# B&R Automation Studio project macie
Automation Studio 4.9

## Configuration Config1

### Hardware
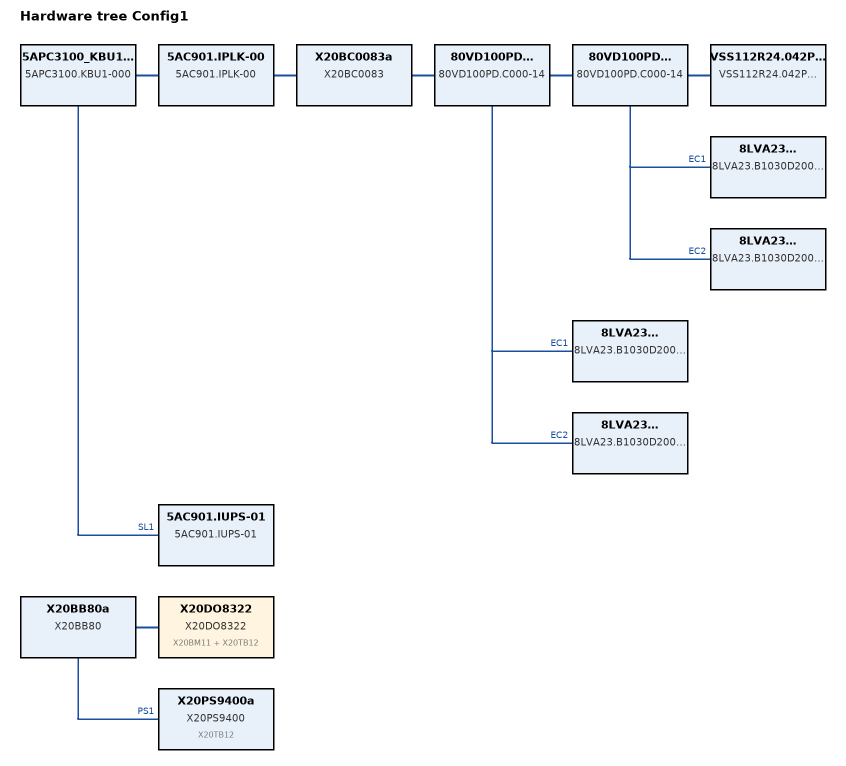
```
5AC901.IPLK-00 : 5AC901.IPLK-00 v1.8.0.1  [SL -> 5APC3100_KBU1_000.SL2]
  Connector IF1:
    MtuSize = 1500
    Channel1
    ChannelID1 = McAcpBroadcast
    ChannelType1 = OCTET[96]
    InternetAddress = 12.10.10.240
    SubnetMask = 255.255.255.0
5AC901.IUPS-01 : 5AC901.IUPS-01 v1.3.1.0  [SL -> 5APC3100_KBU1_000.SL1]
5APC3100_KBU1_000 : 5APC3100.KBU1-000 v2.2.1.0
  Connector IF3:
    AssignedOperatingSystem = ARemb
    ActivateDevice = 1
    Mode = Manual
    InternetAddress = 10.0.0.150
    SubnetMask = 255.255.255.0
    ActivateSnmp = 2
  Connector IF4:
    AssignedOperatingSystem = ARemb
    ActivateDevice = 1
    Mode = Manual
    InternetAddress = 192.168.0.20
    SubnetMask = 255.255.255.0
    ActivateSnmp = 2
  Connector IF5:
    AssignedOperatingSystem = ARemb
  Connector IF6:
    AssignedOperatingSystem = ARemb
  Connector IF7:
    AssignedOperatingSystem = ARemb
  Connector IF8:
    AssignedOperatingSystem = ARemb
  ConfigurationID = prawdziwaDelta_Config1
  Simulation = 1
  TimerDeviceType = EPLX2X
  TimerDevice = 5AC901.IPLK-00.IF1
  TaskClassIdleTime = 2000
  Cyclic1Tolerance = 0
  FileDevice1
  FileDeviceName1 = CNC_PrgDir
  FileDevicePath1 = C:\projects\CNC_PrgDir
  ActivateOpcUa = 1
  OpcUaInformationModels_PV_Version = 1
80VD100PD.C000-14 : 80VD100PD.C000-14 v2.5.0.0  [PLK1 -> X20BC0083a.PLK2 (NodeNumber=1) [Cable Type=PowerlinkCable, Length=10, Version=1.0.0.3]; PLK2 -> 80VD100PD.C000-14a.PLK1 (NodeNumber=1) [Cable Type=PowerlinkCable, Length=10, Version=1.0.0.3]; EC1 -> 8LVA23.B1030D200-0.EC; EC2 -> 8LVA23.B1030D200-0a.EC; MT2 -> 8LVA23.B1030D200-0a.MT]
  DriveConfiguration/Module:
    McAcoposTypeID = AcoposMicroDConfig
    ActivateACOPOSSimulationOnPLC = 0
  DriveConfiguration/Channel[1]/RealAxis:
    AxisReference = gAxisQ1
    MechanicalElementsIsInvisible = 0
  DriveConfiguration/Channel[1]/RealAxis/MechanicalElements/Gearbox:
    InputIsReadOnly = 0
    Input = 25
    OutputIsReadOnly = 0
    Output = 1
  DriveConfiguration/Channel[1]/RealAxis/MechanicalElements/RotaryToLinearTransformation:
    ReferenceDistanceIsReadOnly = 0
    ReferenceDistance = 1
  DriveConfiguration/Channel[1]/RealAxis/Controller:
    ModeIsReadOnly = 0
    Mode = PositionController
  DriveConfiguration/Channel[1]/RealAxis/Controller/Mode/Position:
    ProportionalGain = 402
    IntegrationTime = 0.0
    PredictionTime = 0.0004
    TotalDelayTime = 0.0004
  DriveConfiguration/Channel[1]/RealAxis/Controller/Mode/Speed:
    ProportionalGainIsReadOnly = 0
    ProportionalGain = 1.7
    IntegrationTimeIsReadOnly = 0
    IntegrationTime = 0.0
    FilterTimeIsReadOnly = 0
    FilterTime = 0.0
  DriveConfiguration/Channel[1]/RealAxis/Controller/Mode/LoopFilters:
    LoopFilterXIsReadOnly = 0
    LoopFilter1 = NotUsed
    LoopFilter2 = NotUsed
    LoopFilter3 = NotUsed
  DriveConfiguration/Channel[1]/RealAxis/Homing:
    ModeIsReadOnly = 0
    Mode = Absolute
  DriveConfiguration/Channel[1]/RealAxis/Homing/Mode:
    Position = 0
  DriveConfiguration/Channel[1]/RealAxis/Homing:
    RestorePositionVariable = 
  DriveConfiguration/Channel[1]/RealAxis/StopReaction:
    QuickstopIsReadOnly = 0
    Quickstop = DecelerationLimit
    DriveErrorIsReadOnly = 0
    DriveError = DecelerationLimit
  DriveConfiguration/Channel[1]/RealAxis/MovementErrorLimits:
    PositionError = 1.0
    VelocityErrorMonitoring = Automatic1
  DriveConfiguration/Channel[1]/RealAxis:
    JerkFilterIsReadOnly = 0
    JerkFilter = NotUsed
    ZeroVibrationFilter = NotUsed
  DriveConfiguration/Channel[1]/RealAxis/DigitalInputs/HomingSwitch:
    SourceIsReadOnly = 0
    Source = NotUsed
    Level = High
  DriveConfiguration/Channel[1]/RealAxis/DigitalInputs/PositiveLimitSwitch:
    SourceIsReadOnly = 0
    Source = NotUsed
    Level = High
  DriveConfiguration/Channel[1]/RealAxis/DigitalInputs/NegativeLimitSwitch:
    SourceIsReadOnly = 0
    Source = NotUsed
    Level = High
  DriveConfiguration/Channel[1]/RealAxis/DigitalInputs/Trigger1:
    Source = X2Trigger1
    Level = High
  DriveConfiguration/Channel[1]/RealAxis/DigitalInputs/Trigger2:
    Source = X2Trigger2
    Level = High
  DriveConfiguration/Channel[1]/RealAxis/DigitalInputs/Quickstop:
    Input = Trigger2
  DriveConfiguration/Channel[1]/RealAxis/Simulation:
    SimulationModeOnPLC = SetValueGeneration
    SimulationModeOnACOPOS = NotUsed
  DriveConfiguration/Channel[1]:
    ExternalEncoderAxis = NotUsed
  DriveConfiguration/Channel[2]/RealAxis:
    AxisReference = gAxisQ2
    MechanicalElementsIsInvisible = 0
  DriveConfiguration/Channel[2]/RealAxis/MechanicalElements/Gearbox:
    InputIsReadOnly = 0
    Input = 25
    OutputIsReadOnly = 0
    Output = 1
  DriveConfiguration/Channel[2]/RealAxis/MechanicalElements/RotaryToLinearTransformation:
    ReferenceDistanceIsReadOnly = 0
    ReferenceDistance = 1
  DriveConfiguration/Channel[2]/RealAxis/Controller:
    ModeIsReadOnly = 0
    Mode = PositionController
  DriveConfiguration/Channel[2]/RealAxis/Controller/Mode/Position:
    ProportionalGain = 393
    IntegrationTime = 0.0
    PredictionTime = 0.0004
    TotalDelayTime = 0.0004
  DriveConfiguration/Channel[2]/RealAxis/Controller/Mode/Speed:
    ProportionalGainIsReadOnly = 0
    ProportionalGain = 1.65
    IntegrationTimeIsReadOnly = 0
    IntegrationTime = 0.0
    FilterTimeIsReadOnly = 0
    FilterTime = 0.0
  DriveConfiguration/Channel[2]/RealAxis/Controller/Mode/LoopFilters:
    LoopFilterXIsReadOnly = 0
    LoopFilter1 = NotUsed
    LoopFilter2 = NotUsed
    LoopFilter3 = NotUsed
  DriveConfiguration/Channel[2]/RealAxis/Homing:
    ModeIsReadOnly = 0
    Mode = Absolute
  DriveConfiguration/Channel[2]/RealAxis/Homing/Mode:
    Position = 0
  DriveConfiguration/Channel[2]/RealAxis/Homing:
    RestorePositionVariable = 
  DriveConfiguration/Channel[2]/RealAxis/StopReaction:
    QuickstopIsReadOnly = 0
    Quickstop = DecelerationLimit
    DriveErrorIsReadOnly = 0
    DriveError = DecelerationLimit
  DriveConfiguration/Channel[2]/RealAxis/MovementErrorLimits:
    PositionError = 1.0
    VelocityErrorMonitoring = Automatic1
  DriveConfiguration/Channel[2]/RealAxis:
    JerkFilterIsReadOnly = 0
    JerkFilter = NotUsed
    ZeroVibrationFilter = NotUsed
  DriveConfiguration/Channel[2]/RealAxis/DigitalInputs/HomingSwitch:
    SourceIsReadOnly = 0
    Source = NotUsed
    Level = High
  DriveConfiguration/Channel[2]/RealAxis/DigitalInputs/PositiveLimitSwitch:
    SourceIsReadOnly = 0
    Source = NotUsed
    Level = High
  DriveConfiguration/Channel[2]/RealAxis/DigitalInputs/NegativeLimitSwitch:
    SourceIsReadOnly = 0
    Source = NotUsed
    Level = High
  DriveConfiguration/Channel[2]/RealAxis/DigitalInputs/Trigger1:
    Source = X2Trigger1
    Level = High
  DriveConfiguration/Channel[2]/RealAxis/DigitalInputs/Trigger2:
    Source = X2Trigger2
    Level = High
  DriveConfiguration/Channel[2]/RealAxis/DigitalInputs/Quickstop:
    Input = Trigger2
  DriveConfiguration/Channel[2]/RealAxis/Simulation:
    SimulationModeOnPLC = SetValueGeneration
    SimulationModeOnACOPOS = NotUsed
  DriveConfiguration/Channel[2]:
    ExternalEncoderAxis = NotUsed
80VD100PD.C000-14a : 80VD100PD.C000-14 v2.5.0.0  [PLK1 -> 80VD100PD.C000-14.PLK2 (NodeNumber=2) [Cable Type=PowerlinkCable, Length=10, Version=1.0.0.3]; PLK2 -> VSS112R24.042P-000.PLK1 (NodeNumber=2) [Cable Type=PowerlinkCable, Length=10, Version=1.0.0.3]; EC1 -> 8LVA23.B1030D200-0b.EC; EC2 -> 8LVA23.B1030D200-0c.EC; MT2 -> 8LVA23.B1030D200-0c.MT]
  DriveConfiguration/Module:
    McAcoposTypeID = AcoposMicroDConfig
    ActivateACOPOSSimulationOnPLC = 0
  DriveConfiguration/Channel[1]/RealAxis:
    AxisReference = gAxisQ3
    MechanicalElementsIsInvisible = 0
  DriveConfiguration/Channel[1]/RealAxis/MechanicalElements/Gearbox:
    InputIsReadOnly = 0
    Input = 25
    OutputIsReadOnly = 0
    Output = 1
  DriveConfiguration/Channel[1]/RealAxis/MechanicalElements/RotaryToLinearTransformation:
    ReferenceDistanceIsReadOnly = 0
    ReferenceDistance = 1
  DriveConfiguration/Channel[1]/RealAxis/Controller:
    ModeIsReadOnly = 0
    Mode = PositionController
  DriveConfiguration/Channel[1]/RealAxis/Controller/Mode/Position:
    ProportionalGain = 400
    IntegrationTime = 0.0
    PredictionTime = 0.0004
    TotalDelayTime = 0.0004
  DriveConfiguration/Channel[1]/RealAxis/Controller/Mode/Speed:
    ProportionalGainIsReadOnly = 0
    ProportionalGain = 1.7
    IntegrationTimeIsReadOnly = 0
    IntegrationTime = 0.0
    FilterTimeIsReadOnly = 0
    FilterTime = 0.0
  DriveConfiguration/Channel[1]/RealAxis/Controller/Mode/LoopFilters:
    LoopFilterXIsReadOnly = 0
    LoopFilter1 = NotUsed
    LoopFilter2 = NotUsed
    LoopFilter3 = NotUsed
  DriveConfiguration/Channel[1]/RealAxis/Homing:
    ModeIsReadOnly = 0
    Mode = Absolute
  DriveConfiguration/Channel[1]/RealAxis/Homing/Mode:
    Position = 0
  DriveConfiguration/Channel[1]/RealAxis/Homing:
    RestorePositionVariable = 
  DriveConfiguration/Channel[1]/RealAxis/StopReaction:
    QuickstopIsReadOnly = 0
    Quickstop = DecelerationLimit
    DriveErrorIsReadOnly = 0
    DriveError = DecelerationLimit
  DriveConfiguration/Channel[1]/RealAxis/MovementErrorLimits:
    PositionError = 1.0
    VelocityErrorMonitoring = Automatic1
  DriveConfiguration/Channel[1]/RealAxis:
    JerkFilterIsReadOnly = 0
    JerkFilter = NotUsed
    ZeroVibrationFilter = NotUsed
  DriveConfiguration/Channel[1]/RealAxis/DigitalInputs/HomingSwitch:
    SourceIsReadOnly = 0
    Source = NotUsed
    Level = High
  DriveConfiguration/Channel[1]/RealAxis/DigitalInputs/PositiveLimitSwitch:
    SourceIsReadOnly = 0
    Source = NotUsed
    Level = High
  DriveConfiguration/Channel[1]/RealAxis/DigitalInputs/NegativeLimitSwitch:
    SourceIsReadOnly = 0
    Source = NotUsed
    Level = High
  DriveConfiguration/Channel[1]/RealAxis/DigitalInputs/Trigger1:
    Source = X2Trigger1
    Level = High
  DriveConfiguration/Channel[1]/RealAxis/DigitalInputs/Trigger2:
    Source = X2Trigger2
    Level = High
  DriveConfiguration/Channel[1]/RealAxis/DigitalInputs/Quickstop:
    Input = Trigger2
  DriveConfiguration/Channel[1]/RealAxis/Simulation:
    SimulationModeOnPLC = SetValueGeneration
    SimulationModeOnACOPOS = NotUsed
  DriveConfiguration/Channel[1]:
    ExternalEncoderAxis = NotUsed
  DriveConfiguration/Channel[2]/RealAxis:
    AxisReference = gAxis_1
    MechanicalElementsIsInvisible = 0
  DriveConfiguration/Channel[2]/RealAxis/MechanicalElements/Gearbox:
    InputIsReadOnly = 0
    Input = 1
    OutputIsReadOnly = 0
    Output = 1
  DriveConfiguration/Channel[2]/RealAxis/MechanicalElements/RotaryToLinearTransformation:
    ReferenceDistanceIsReadOnly = 0
    ReferenceDistance = 1
  DriveConfiguration/Channel[2]/RealAxis/Controller:
    ModeIsReadOnly = 0
    Mode = PositionController
  DriveConfiguration/Channel[2]/RealAxis/Controller/Mode/Position:
    ProportionalGain = 50.0
    IntegrationTime = 0.0
    PredictionTime = 0.0004
    TotalDelayTime = 0.0004
  DriveConfiguration/Channel[2]/RealAxis/Controller/Mode/Speed:
    ProportionalGainIsReadOnly = 0
    ProportionalGain = 2.0
    IntegrationTimeIsReadOnly = 0
    IntegrationTime = 0.0
    FilterTimeIsReadOnly = 0
    FilterTime = 0.0
  DriveConfiguration/Channel[2]/RealAxis/Controller/Mode/LoopFilters:
    LoopFilterXIsReadOnly = 0
    LoopFilter1 = NotUsed
    LoopFilter2 = NotUsed
    LoopFilter3 = NotUsed
  DriveConfiguration/Channel[2]/RealAxis/Homing:
    ModeIsReadOnly = 0
    Mode = Direct
  DriveConfiguration/Channel[2]/RealAxis/Homing/Mode:
    Position = 0.0
    ReferencePulse = NotUsed
  DriveConfiguration/Channel[2]/RealAxis/Homing:
    RestorePositionVariable = 
  DriveConfiguration/Channel[2]/RealAxis/StopReaction:
    QuickstopIsReadOnly = 0
    Quickstop = DecelerationLimit
    DriveErrorIsReadOnly = 0
    DriveError = DecelerationLimit
  DriveConfiguration/Channel[2]/RealAxis/MovementErrorLimits:
    PositionError = 1.0
    VelocityErrorMonitoring = Automatic1
  DriveConfiguration/Channel[2]/RealAxis:
    JerkFilterIsReadOnly = 0
    JerkFilter = NotUsed
    ZeroVibrationFilter = NotUsed
  DriveConfiguration/Channel[2]/RealAxis/DigitalInputs/HomingSwitch:
    SourceIsReadOnly = 0
    Source = NotUsed
    Level = High
  DriveConfiguration/Channel[2]/RealAxis/DigitalInputs/PositiveLimitSwitch:
    SourceIsReadOnly = 0
    Source = NotUsed
    Level = High
  DriveConfiguration/Channel[2]/RealAxis/DigitalInputs/NegativeLimitSwitch:
    SourceIsReadOnly = 0
    Source = NotUsed
    Level = High
  DriveConfiguration/Channel[2]/RealAxis/DigitalInputs/Trigger1:
    Source = X2Trigger1
    Level = High
  DriveConfiguration/Channel[2]/RealAxis/DigitalInputs/Trigger2:
    Source = X2Trigger2
    Level = High
  DriveConfiguration/Channel[2]/RealAxis/DigitalInputs/Quickstop:
    Input = Trigger2
  DriveConfiguration/Channel[2]/RealAxis/Simulation:
    SimulationModeOnPLC = SetValueGeneration
    SimulationModeOnACOPOS = NotUsed
  DriveConfiguration/Channel[2]:
    ExternalEncoderAxis = NotUsed
8LVA23.B1030D200-0 : 8LVA23.B1030D200-0 v2.2.0.3  [EC -> 80VD100PD.C000-14.EC1; MT -> 80VD100PD.C000-14.MT1]
  M1/MotorParameters:
    MOTOR_AMB_TEMP_RATED = 40
8LVA23.B1030D200-0a : 8LVA23.B1030D200-0 v2.2.0.3  [EC -> 80VD100PD.C000-14.EC2; MT -> 80VD100PD.C000-14.MT2]
  M1/MotorParameters:
    MOTOR_AMB_TEMP_RATED = 40
8LVA23.B1030D200-0b : 8LVA23.B1030D200-0 v2.2.0.3  [EC -> 80VD100PD.C000-14a.EC1; MT -> 80VD100PD.C000-14a.MT1]
  M1/MotorParameters:
    MOTOR_AMB_TEMP_RATED = 40
8LVA23.B1030D200-0c : 8LVA23.B1030D200-0 v2.2.0.3  [EC -> 80VD100PD.C000-14a.EC2; MT -> 80VD100PD.C000-14a.MT2]
  M1/MotorParameters:
    MOTOR_AMB_TEMP_RATED = 40
VSS112R24.042P-000 : VSS112R24.042P-000 v1.9.0.730  [PLK1 -> 80VD100PD.C000-14a.PLK2 (NodeNumber=4) [Cable Type=PowerlinkCable, Length=10, Version=1.0.0.3]]
  Supervision = off
  VisionConfig = gCamera
X20BB80a : X20BB80 v1.1.0.0
X20BC0083a : X20BC0083 v2.14.0.0  [PLK1 -> 5AC901.IPLK-00.IF1 (NodeNumber=3) [Cable Type=PowerlinkCable, Length=10, Version=1.0.0.3]; PLK2 -> 80VD100PD.C000-14.PLK1 (NodeNumber=3) [Cable Type=PowerlinkCable, Length=10, Version=1.0.0.3]; SL -> X20BB80a.SL1]
  Supervision = off
X20BM11a : X20BM11 v1.1.0.0  [X2X1 -> X20BB80a.IF1]
X20DO8322 : X20DO8322 v1.5.0.0  [SS1 -> X20TB12b.SS; SL -> X20BM11a.SL1]
X20PS9400a : X20PS9400 v1.8.0.0  [SS1 -> X20TB12a.SS; PS -> X20BB80a.PS1]
  Supervision = off
X20TB12a : X20TB12 v1.0.0.0
X20TB12b : X20TB12 v1.0.0.0
```

### Config_8.pickregister - 5APC3100_KBU1_000/mappMotion/Config_8.pickregister
```
Element gPickRegister (Type=pickregister)
  Type = LinearConveyor
    StandardFrameName = ConveyorPick
    Length = 600
    Width = 120
    Height = 6
    MaxPositionError = 10
    MotionSource = Axis
      AxisRef = gAxis_1
      MovementLimits = UseAxisLimits
        Direction = Bidirectional
  SceneViewerObject = Used
    VisualRepresentation = Conveyor belt
      Dimensions:
        Length = 0.0
        Width = 0.0
        Height = 0.0
      Translation:
        X = 0.0
        Y = 0.0
        Z = 0.0
      Orientation:
        Angle1 = 0.0
        Angle2 = 0.0
        Angle3 = 0.0
    Content:
      Template[1]:
        VisualRepresentation = 2DShape
          ShapeType:
            Dimensions:
              Radius = 25.0
            Translation:
              X = 0.0
              Y = 0.0
              Z = 0.0
            Orientation:
              Angle1 = 0.0
              Angle2 = 0.0
              Angle3 = 0.0
        Filter:
          ObjectState:
            State[1] = 1
      Template[2]:
        VisualRepresentation:
          Size = 50.0
        Filter:
          ObjectState:
            State[1] = 2
  Alarms = None
Element gPlaceRegister (Type=pickregister)
  Type = LinearConveyor
    StandardFrameName = ConveyorPlace
    Length = 215
    Width = 60
    Height = 10
    MaxItems = 5
    MaxPositionError = 10
    MotionSource = Axis
      AxisRef = gAxis_2
      MovementLimits = UseAxisLimits
        Direction = Bidirectional
  SceneViewerObject = Used
    VisualRepresentation = Cuboid
      Dimensions:
        Length = 215
        Width = 60
        Height = 50
      Translation:
        X = 0.0
        Y = 0.0
        Z = 0.0
      Orientation:
        Angle1 = 0.0
        Angle2 = 0.0
        Angle3 = 0.0
    Content:
      Template[1]:
        VisualRepresentation = 2DShape
          ShapeType:
            Dimensions:
              Radius = 25.0
            Translation:
              X = 0.0
              Y = 0.0
              Z = 0.0
            Orientation:
              Angle1 = 0.0
              Angle2 = 0.0
              Angle3 = 0.0
        Filter:
          ObjectState:
            State[1] = 1
      Template[2]:
        VisualRepresentation:
          Size = 50.0
        Filter:
          ObjectState:
            State[1] = 1
  Alarms = None
```

## Logical view

### Robotic.st
```iecst
VAR CONSTANT
P1 : McPointType := (Pos:=(X:=0, Y:=0, Z:=-650));
P2 : McPointType := (Pos:=(X:=-50, Y:=-20, Z:=-600));
P0 : McPointType := (Pos:=(X:=0, Y:=0, Z:=-560));
	END_VAR

	PROGRAM _MAIN
	Feedrate(5000);   //move with reduced speed
	MoveJ(P1);        //move system to point P1
	MoveJ(P2);        //move system to point P2

	WaitTime(3);        //wait for 3 seconds

	MoveJ(P0);        //move back to origin position
	END_PROGRAM
```

### Program Logical/PickAndPlace/PrgMechs (IEC) - Handle Delta & Conveyor Belts

#### Main.st
```iecst
PROGRAM _INIT

	MpDelta4Axis_0.Override := 100.0;
	MpDelta4Axis_0.Enable   := TRUE;

	AxisParameters_0.Velocity     := 50.0;
	AxisParameters_0.Acceleration := 50.0;
	AxisParameters_0.Deceleration := 50.0;

	AxisParameters_1.Velocity     := 130.0;
	AxisParameters_1.Acceleration := 50.0;
	AxisParameters_1.Deceleration := 50.0;

	MpAxisBasic_0.Enable := TRUE;
	MpAxisBasic_1.Enable := TRUE;

	// dummy call of axis PVs just to avoid warning -2141192189 "The PV 'gAxisQx' does not exists" in logger
	gAxisQ1;
	gAxisQ2;
	gAxisQ3;
	gAxisQ4;

END_PROGRAM

PROGRAM _CYCLIC

    (* Prepare mechanics: Robot & conveyors *)
	CASE RC_Step OF

		(* first preparing robot *)
		RC_WAIT_ENABLE:
			IF MpDelta4Axis_0.Active THEN
				RC_Step := RC_POWER_ROBOT;
			END_IF

		RC_POWER_ROBOT:
			MpDelta4Axis_0.Power := TRUE;
			IF MpDelta4Axis_0.PowerOn THEN
				RC_Step := RC_HOME_ROBOT;
			END_IF

		RC_HOME_ROBOT:
			MpDelta4Axis_0.Home := TRUE;
			IF MpDelta4Axis_0.IsHomed THEN
				MpDelta4Axis_0.Home := FALSE;
				RC_Step := RC_ROBOT_READY;
			END_IF

		RC_ROBOT_READY:
			RC_Step := RC_WAIT_ENABLE_AXIS_FB;

			(* preparing conveyors *)
		RC_WAIT_ENABLE_AXIS_FB:
			IF MpAxisBasic_0.Active THEN
				IF MpAxisBasic_1.Active THEN
					RC_Step := RC_POWER_AXIS;
				END_IF
			ELSIF MpAxisBasic_0.Error  THEN
				LastStep := RC_Step;
				RC_Step  := RC_ERROR;
			END_IF;

		RC_POWER_AXIS:
			MpAxisBasic_0.Power := TRUE;
			MpAxisBasic_1.Power := TRUE;
			RC_Step := RC_WAIT_POWER_AXIS;

		RC_WAIT_POWER_AXIS:
			IF MpAxisBasic_0.PowerOn THEN
				IF MpAxisBasic_1.PowerOn THEN
					RC_Step := RC_HOME_AXIS;
				END_IF
			ELSIF MpAxisBasic_0.Error  THEN
				LastStep := RC_Step;
				RC_Step  := RC_ERROR;
			END_IF;

		RC_HOME_AXIS:
			MpAxisBasic_0.Home := TRUE;
			MpAxisBasic_1.Home := TRUE;
			RC_Step := RC_WAIT_HOME_AXIS;

		RC_WAIT_HOME_AXIS:
			IF MpAxisBasic_0.IsHomed THEN
				IF MpAxisBasic_0.IsHomed THEN
					MpAxisBasic_0.Home := FALSE;
					MpAxisBasic_1.Home := FALSE;
					RC_Step := RC_READY;
				END_IF
			ELSIF MpAxisBasic_0.Error  THEN
				LastStep := RC_Step;
				RC_Step  := RC_ERROR;
			END_IF;

		RC_READY:
			ReadyMechanics := TRUE;
			IF CmdStart AND ReadyToStart THEN
				RC_Step := RC_START_PROCESS;
			END_IF;

			(* start conveyors to move *)
		RC_START_PROCESS:
			MpAxisBasic_0.MoveVelocity := TRUE;
			//  MpAxisBasic_1.MoveVelocity := TRUE;
			RC_Step := RC_WAIT_PROCESS_STARTED;

		RC_WAIT_PROCESS_STARTED:
			IF MpAxisBasic_0.Info.PLCopenState = mcAXIS_CONTINUOUS_MOTION THEN
				//   IF MpAxisBasic_1.Info.PLCopenState = mcAXIS_CONTINUOUS_MOTION THEN
				RC_Step := RC_PROCESSING;
				//  END_IF
			ELSIF MpAxisBasic_0.Error  THEN
				LastStep := RC_Step;
				RC_Step  := RC_ERROR;
			END_IF;

		RC_PROCESSING:
			IF MpAxisBasic_0.Error  THEN
				LastStep := RC_Step;
				RC_Step  := RC_ERROR;
			END_IF;

		RC_ERROR:
			ReadyMechanics := FALSE;

	END_CASE

	ReadyToStart := ReadyMechanics AND ReadyPickReg AND ReadyPlaceReg AND ReadyPickCore;

	(* Call FBs *)
	MpDelta4Axis_0.MpLink     := ADR(g4AxDeltaA);
	MpDelta4Axis_0.Parameters := ADR(DeltaParameters);
	MpDelta4Axis_0();

	MpAxisBasic_0.MpLink     := ADR(gAxis_1);
	MpAxisBasic_0.Parameters := ADR(AxisParameters_0);
	MpAxisBasic_0();

	MpAxisBasic_1.MpLink     := ADR(gAxis_2);
	MpAxisBasic_1.Parameters := ADR(AxisParameters_1);
	MpAxisBasic_1();

	PickConveyorPosition  := MpAxisBasic_0.Position;
	PlaceConveyorPosition := MpAxisBasic_1.Position;

END_PROGRAM
```

### Program Logical/PickAndPlace/PrgPlace (IEC) - Place the products

#### Types.typ
```iecst
TYPE
	PlaceStepEnum :
		(
		P_WAIT_ENABLE,
		P_ENABLE_REGISTER_FB,
		P_WAIT_ENABLE_REGISTER_FB,
		P_ENABLE_REGISTER_COMP,
		P_WAIT_ENABLE_REGISTER_COMP,
		P_ENABLE_ADD_REGISTER_FBS,
		P_WAIT_ENABLE_ADD_REGISTER_FBS,
		P_WAIT_START_PROCESS,
		P_CREATE_OBJECTS,
		P_WAIT_CREATE_OBJECTS,
		P_WAIT_REGISTER_FULL,
		P_DELAY_DELETE,
		P_DELETE_OBJECTS,
		P_WAIT_DELETE_OBJECTS,
		P_DELAY_CREATE,
		P_ERROR
	);
END_TYPE
```

#### Variables.var
```iecst
VAR
	P_Step : PlaceStepEnum;
	LastStep : PlaceStepEnum;
	Error : BOOL;
	PlaceHoldersSpacing : LREAL;
	LastPlaceHolderConveyorPosition : LREAL;
	ElapsedDistance : LREAL;
END_VAR
(*   *)
(*Functionblocks*)
VAR
	MpPickRegCreatePlaceholder1 : MpPickRegCreateObject;
	MpPickRegCreatePlaceholder2 : MpPickRegCreateObject;
	MpPickRegCreatePlaceholder3 : MpPickRegCreateObject;
	MpPickRegCreatePlaceholder : MpPickRegCreateObject;
	MpPickRegister_0 : MpPickRegister;
	polka : USINT;
	tablicaPlace : ARRAY[0..3] OF LREAL;
	PlaceY : LREAL;
	iteracja : INT;
	abc : BOOL;
END_VAR
```

#### Main.st
```iecst
PROGRAM _INIT

	P_Step := P_WAIT_ENABLE;
	Error := FALSE;
	restart := FALSE;
	polka := 0;
	PlaceHoldersSpacing := 120; // distance between two consecutive place holders
	tablicaPlace[0] := 4;
	tablicaPlace[1] := 48;
	tablicaPlace[2] := 96;
	tablicaPlace[3] := 144;

	PlaceY := 30;

	abc := 0;
	iteracja := 0;
END_PROGRAM

PROGRAM _CYCLIC

	CASE P_Step OF
		P_WAIT_ENABLE:
			P_Step := P_ENABLE_REGISTER_FB;

		P_ENABLE_REGISTER_FB:
			MpPickRegister_0.Enable := TRUE;
			P_Step := P_WAIT_ENABLE_REGISTER_FB;

		P_WAIT_ENABLE_REGISTER_FB:
			IF MpPickRegister_0.Active THEN
				P_Step := P_ENABLE_REGISTER_COMP;

			ELSIF MpPickRegister_0.Error THEN
				LastStep := P_Step;
				P_Step := P_ERROR;
			END_IF;

		P_ENABLE_REGISTER_COMP:
			MpPickRegister_0.RegisterEnable := TRUE;
			P_Step := P_WAIT_ENABLE_REGISTER_COMP;

		P_WAIT_ENABLE_REGISTER_COMP:
			IF MpPickRegister_0.RegisterActive THEN
				P_Step := P_ENABLE_ADD_REGISTER_FBS;

			ELSIF MpPickRegister_0.Error THEN
				LastStep := P_Step;
				P_Step := P_ERROR;
			END_IF;

		P_ENABLE_ADD_REGISTER_FBS:
			MpPickRegCreatePlaceholder.Enable := TRUE;
			MpPickRegCreatePlaceholder.Create := FALSE;
			P_Step := P_WAIT_ENABLE_ADD_REGISTER_FBS;

		P_WAIT_ENABLE_ADD_REGISTER_FBS:
			IF 	MpPickRegCreatePlaceholder.Active THEN
				P_Step := P_WAIT_START_PROCESS;

			ELSIF MpPickRegCreatePlaceholder.Error THEN
				LastStep := P_Step;
				P_Step := P_ERROR;
			END_IF;

		P_WAIT_START_PROCESS: // waits user start command and conveyor moving
			ReadyPlaceReg := TRUE;
			IF CmdStart AND ReadyToStart (*AND (PlaceConveyorPosition > 0)*) THEN
				P_Step := P_CREATE_OBJECTS;
			END_IF;

			(* We need to create positions (place holders) on place conveyor where to place picked objects *)
		P_CREATE_OBJECTS:

			IF abc THEN

				CASE iteracja OF
					0:
						MpPickRegCreatePlaceholder.Parameters.LatchedConveyor.Position := PlaceConveyorPosition;
						MpPickRegCreatePlaceholder.Parameters.Mode := mpPICK_CREATE_SINGLEITEM_PLACEH;
						MpPickRegCreatePlaceholder.Parameters.ObjectTypeName := 'MyProduct';
						MpPickRegCreatePlaceholder.Parameters.Translation.X := tablicaPlace[0];
						MpPickRegCreatePlaceholder.Parameters.Translation.Y := PlaceY; // in the middle of conveyor width
						MpPickRegCreatePlaceholder.Create := TRUE;
						iteracja := 1;
						abc := 0;

					1:
						MpPickRegCreatePlaceholder.Parameters.LatchedConveyor.Position := PlaceConveyorPosition;
						MpPickRegCreatePlaceholder.Parameters.Mode := mpPICK_CREATE_SINGLEITEM_PLACEH;
						MpPickRegCreatePlaceholder.Parameters.ObjectTypeName := 'MyProduct';
						MpPickRegCreatePlaceholder.Parameters.Translation.X := tablicaPlace[1];
						MpPickRegCreatePlaceholder.Parameters.Translation.Y := PlaceY; // in the middle of conveyor width
						MpPickRegCreatePlaceholder.Create := TRUE;
						iteracja := 2;
						abc := 0;
					2:
						MpPickRegCreatePlaceholder.Parameters.LatchedConveyor.Position := PlaceConveyorPosition;
						MpPickRegCreatePlaceholder.Parameters.Mode := mpPICK_CREATE_SINGLEITEM_PLACEH;
						MpPickRegCreatePlaceholder.Parameters.ObjectTypeName := 'MyProduct';
						MpPickRegCreatePlaceholder.Parameters.Translation.X := tablicaPlace[2];
						MpPickRegCreatePlaceholder.Parameters.Translation.Y := PlaceY; // in the middle of conveyor width
						MpPickRegCreatePlaceholder.Create := TRUE;
						iteracja := 3;
						abc := 0;

					3:
						MpPickRegCreatePlaceholder.Parameters.LatchedConveyor.Position := PlaceConveyorPosition;
						MpPickRegCreatePlaceholder.Parameters.Mode := mpPICK_CREATE_SINGLEITEM_PLACEH;
						MpPickRegCreatePlaceholder.Parameters.ObjectTypeName := 'MyProduct';
						MpPickRegCreatePlaceholder.Parameters.Translation.X := tablicaPlace[3];
						MpPickRegCreatePlaceholder.Parameters.Translation.Y := PlaceY; // in the middle of conveyor width
						MpPickRegCreatePlaceholder.Create := TRUE;
						iteracja := 4;
						abc := 0;
					4:
						abc :=0;
				END_CASE;
			ELSE
				MpPickRegCreatePlaceholder.Create := FALSE;
				abc :=1;
			END_IF

		P_ERROR:
			Error := TRUE;
			ReadyPlaceReg := FALSE;

	END_CASE;

	(* FB calls *)
	MpPickRegister_0.MpLink := ADR(gPlaceRegister);
	MpPickRegister_0();

	MpPickRegCreatePlaceholder.MpLink := ADR(gPlaceRegister);
	MpPickRegCreatePlaceholder();

END_PROGRAM
```

### Program Logical/PickAndPlace/Program (IEC)

#### Types.typ
```iecst
TYPE
	Krok :
		(
		HOME,
		POWER,
		PROG,
		CHECK,
		RUCH,
		FLAGI,
		WAIT
		);
END_TYPE
```

Listed in the project but not available here: Logical/PickAndPlace/UserLibraries, Logical/PickAndPlace/PrgGlobal.var, Logical/PickAndPlace/PrgPickCore, Logical/PickAndPlace/PrgPick, Logical/PickAndPlace/Scene, Logical/PickAndPlace/TCPXYZ
